PROGRAM MAIN
VAR
	//strategy controller
	Strategy : FB_BaseStrategyController; 

	//thermal networks
	CN : FB_CoolingNetwork;
	HNLT_CN : FB_HnltCnLinkage;
	HNLT : FB_LowTemperatureHeatingNetwork;
	
	//ambient state
	Ambient : FB_Ambient;
END_VAR

//strategy controller
Strategy(stAmbientState := Ambient.stAmtbientState,
	fTemperature_CN := CN.fTemperatureBufferStorage,
	fTemperature_HNLT := HNLT.fTemperatureBufferStorage);

//ambient state
Ambient();
	
//thermal networks
CN(stCNControl := Strategy.stCNControl);

HNLT_CN(stHnltCnLinkageControl := Strategy.stHnltCnLinkageControl);
	
HNLT(stAmbientState := Ambient.stAmtbientState,
	stHNLTControl := Strategy.stHNLTControl);

END_PROGRAM

(* stored: Version 1.1.0.1, ProductVersion 3.1.4024.10
   POU MAIN: Id {9f33f5a0-2a24-4206-9468-c589128c5602}, SpecialFunc None *)
